{attribute 'linkalways'} 
{attribute 'no_explicit_call' := 'This FB is a CLASS and must be accessed using methods or properties'}
{attribute 'enable_dynamic_creation'}
FUNCTION_BLOCK _DWORD EXTENDS NumericDatatypeBase implements I_DWORD
VAR
	localData : DWORD;
	activeData : REFERENCE TO DWORD REF= localData;
END_VAR

PROPERTY PUBLIC Address : PVOID
GET
Address := ADR(activeData);
END_GET
END_PROPERTY

METHOD PUBLIC ClearReference
VAR_INPUT
END_VAR
activeData REF= localData;
END_METHOD

METHOD PUBLIC Clone : I_Datatype
VAR
    pClone : POINTER TO _DWORD;
END_VAR
pClone := __NEW(_DWORD(InitialValue := Value));
Clone := pClone^;
END_METHOD

METHOD FB_init : BOOL
VAR_INPUT
	bInitRetains : BOOL; // if TRUE, the retain variables are initialized (warm start / cold start)
	bInCopyCode : BOOL;  // if TRUE, the instance afterwards gets moved WORDo the copy code (online change)
	InitialValue : DWORD;
END_VAR
localData := InitialValue;
END_METHOD

PROPERTY PUBLIC IsEven : BOOL
GET
IsEven := (Value mod 2) = 0;
END_GET
END_PROPERTY

PROPERTY PUBLIC IsFloat : BOOL
GET
IsFloat := FALSE;
END_GET
END_PROPERTY

PROPERTY PUBLIC IsSigned : BOOL
GET
IsSigned := FALSE;
END_GET
END_PROPERTY

METHOD PUBLIC MakeReferenceTo
VAR_INPUT
	ReferenceTarget : REFERENCE TO DWORD;
END_VAR
activeData REF= ReferenceTarget;
END_METHOD

PROPERTY PUBLIC MaxValue : DWORD
GET
MaxValue := DatatypeLimits.DWORD_MAX_VALUE;
END_GET
END_PROPERTY

PROPERTY PUBLIC MinValue : DWORD
GET
MinValue := DatatypeLimits.DWORD_MIN_VALUE;
END_GET
END_PROPERTY

METHOD PROTECTED SerializeMaxValue
VAR_INPUT
	Serializer : I_Serializer;
END_VAR
Serializer.AddDword(MaxValue);
END_METHOD

METHOD PROTECTED SerializeMinValue
VAR_INPUT
	Serializer : I_Serializer;
END_VAR
Serializer.AddDword(MinValue);
END_METHOD

METHOD PUBLIC SerializeWith
VAR_INPUT
	Serializer : I_Serializer;
END_VAR
Serializer.AddDword(activeData);
END_METHOD

PROPERTY PUBLIC Size : UDINT
GET
Size := SIZEOF(activeData);
END_GET
END_PROPERTY

METHOD PUBLIC TryConvertTo : BOOL
VAR_INPUT
	Destination : ANY;
END_VAR
TryConvertTo := TryConvert_DWORD_To_Destination(activeData, Destination);
END_METHOD

METHOD PUBLIC TryConvertTo_ : BOOL
VAR_INPUT
	Destination : I_Datatype;
END_VAR
VAR
	resultofBitConversion : BOOL;
	destinationAs_BIT : I_BIT;
	destinationAs_BOOL : I_BOOL;
	destinationAs_BYTE : I_BYTE;
	destinationAs_DINT : I_DINT;
	destinationAs_DT : I_DT;
	destinationAs_DWORD : I_DWORD;
	destinationAs_INT : I_INT;
	destinationAs_LINT : I_LINT;
	destinationAs_LREAL : I_LREAL;
	destinationAs_LWORD : I_LWORD;
	destinationAs_REAL : I_REAL;
	destinationAs_SINT : I_SINT;
	destinationAs_STRING : I_STRING;
	destinationAs_TOD : I_TOD;
	destinationAs_UDINT : I_UDINT;
	destinationAs_UINT : I_UINT;
	destinationAs_ULINT : I_ULINT;
	destinationAs_USINT : I_USINT;
	destinationAs_WORD : I_WORD;
END_VAR
IF destination.TryResolveAs_BIT(destinationAs_BIT) AND_THEN TryConvert_DWORD_TO_BOOL(activeData, resultofBitConversion) THEN
	destinationAs_BIT.Value := resultOfBitConversion;
	TryConvertTo_ := TRUE;
	RETURN;
END_IF

IF destination.TryResolveAs_BOOL(destinationAs_BOOL) THEN
	TryConvertTo_ := TryConvert_DWORD_TO_BOOL(activeData, destinationAs_BOOL.Value);
	RETURN;
END_IF
		
IF destination.TryResolveAs_BYTE(destinationAs_BYTE) THEN
	TryConvertTo_ := TryConvert_DWORD_TO_BYTE(activeData, destinationAs_BYTE.Value);
	RETURN;
END_IF

IF destination.TryResolveAs_DINT(destinationAs_DINT) THEN
	TryConvertTo_ := TryConvert_DWORD_TO_DINT(activeData, destinationAs_DINT.Value);
	RETURN;
END_IF

IF destination.TryResolveAs_DT(destinationAs_DT) THEN
	TryConvertTo_ := TryConvert_DWORD_TO_DT(activeData, destinationAs_DT.Value);
	RETURN;
END_IF

IF destination.TryResolveAs_DWORD(destinationAs_DWORD) THEN
	TryConvertTo_ := TryConvert_DWORD_TO_DWORD(activeData, destinationAs_DWORD.Value);
	RETURN;
END_IF

IF destination.TryResolveAs_INT(destinationAs_INT) THEN
	TryConvertTo_ := TryConvert_DWORD_TO_INT(activeData, destinationAs_INT.Value);
	RETURN;
END_IF

IF destination.TryResolveAs_LINT(destinationAs_LINT) THEN
	TryConvertTo_ := TryConvert_DWORD_TO_LINT(activeData, destinationAs_LINT.Value);
	RETURN;
END_IF

IF destination.TryResolveAs_LREAL(destinationAs_LREAL) THEN
	TryConvertTo_ := TryConvert_DWORD_TO_LREAL(activeData, destinationAs_LREAL.Value);
	RETURN;
END_IF

IF destination.TryResolveAs_LWORD(destinationAs_LWORD) THEN
	TryConvertTo_ := TryConvert_DWORD_TO_LWORD(activeData, destinationAs_LWORD.Value);
	RETURN;
END_IF

IF destination.TryResolveAs_REAL(destinationAs_REAL) THEN
	TryConvertTo_ := TryConvert_DWORD_TO_REAL(activeData, destinationAs_REAL.Value);
	RETURN;
END_IF

IF destination.TryResolveAs_SINT(destinationAs_SINT) THEN
	TryConvertTo_ := TryConvert_DWORD_TO_SINT(activeData, destinationAs_SINT.Value);
	RETURN;
END_IF

IF destination.TryResolveAs_STRING(destinationAs_STRING) THEN
	TryConvertTo_ := TryConvert_DWORD_TO_STRING(activeData, destinationAs_STRING.Value);
	RETURN;
END_IF

IF destination.TryResolveAs_TOD(destinationAs_TOD) THEN
	TryConvertTo_ := TryConvert_DWORD_TO_TOD(activeData, destinationAs_TOD.Value);
	RETURN;
END_IF

IF destination.TryResolveAs_UDINT(destinationAs_UDINT) THEN
	TryConvertTo_ := TryConvert_DWORD_TO_UDINT(activeData, destinationAs_UDINT.Value);
	RETURN;
END_IF

IF destination.TryResolveAs_UINT(destinationAs_UINT) THEN
	TryConvertTo_ := TryConvert_DWORD_TO_UINT(activeData, destinationAs_UINT.Value);
	RETURN;
END_IF

IF destination.TryResolveAs_ULINT(destinationAs_ULINT) THEN
	TryConvertTo_ := TryConvert_DWORD_TO_ULINT(activeData, destinationAs_ULINT.Value);
	RETURN;
END_IF

IF destination.TryResolveAs_USINT(destinationAs_USINT) THEN
	TryConvertTo_ := TryConvert_DWORD_TO_USINT(activeData, destinationAs_USINT.Value);
	RETURN;
END_IF

IF destination.TryResolveAs_WORD(destinationAs_WORD) THEN
	TryConvertTo_ := TryConvert_DWORD_TO_WORD(activeData, destinationAs_WORD.Value);
	RETURN;
END_IF
END_METHOD

METHOD TryDeserializeFrom : BOOL
VAR_INPUT
	Deserializer : I_Deserializer;
	Feedback : I_DeserializerFeedback;
END_VAR
TryDeserializeFrom := Deserializer.TryGetDword(activeData, Feedback);
END_METHOD

METHOD TryMakeReferenceTo : BOOL
VAR_INPUT
	Target : I_Datatype;
END_VAR
VAR
	pTargetData : POINTER TO DWORD;
END_VAR
IF NOT IsEquivalentTo(Target) THEN
	RETURN;
END_IF

pTargetData := Target.Address;
activeData REF= pTargetData^;
TryMakeReferenceTo := TRUE;
END_METHOD

METHOD PUBLIC TryResolveAs_DWORD : BOOL
VAR_INPUT
	Destination : REFERENCE TO I_DWORD;
END_VAR
Destination := THIS^;
TryResolveAs_DWORD := TRUE;
END_METHOD

PROPERTY PUBLIC TypeName : T_MAXSTRING
GET
TypeName := 'DWORD';
END_GET
END_PROPERTY

PROPERTY PUBLIC Value : REFERENCE TO DWORD
GET
Value REF= activeData;
END_GET
END_PROPERTY

END_FUNCTION_BLOCK

(* stored: Version 1.1.0.1, ProductVersion 3.1.4024.15
   POU _DWORD: Id {0e1f4684-9ced-429c-808b-7eae4b4c544d}, SpecialFunc None
   Folder Constructor: Id {ed0f11a9-1e9f-4982-8f38-38243a563b64}
   Folder Protected: Id {81979a9d-08ab-4990-a6a1-6d8257d387e2}
   Property Address: Id {db5664d4-745e-4039-a24f-c4ccfecba779}
   Get Get: Id {e031636d-09ee-4c01-a84d-b6877667d967}
   Method ClearReference: Id {d4461140-18cc-4879-b0d4-8191674e6247}
   Method Clone: Id {94d3bddf-8fcb-4938-8fbd-23c2da87ed5a}
   Method FB_init: Id {12a44695-f484-4b13-adf1-9bfc8d3ddbe4}
   Property IsEven: Id {a9233086-77fa-0502-3db7-4b000f1aa9c4}
   Get Get: Id {42c8b3e7-f556-0983-013b-60f8adaee327}
   Property IsFloat: Id {ad06f207-ab0a-4f8c-a31f-a02263d34b51}
   Get Get: Id {203ea2a5-3922-43d2-862b-de05e5f89dd5}
   Property IsSigned: Id {513f9891-7111-4f35-92cb-cbc81f2c7472}
   Get Get: Id {8417e378-9fc5-4222-8e5d-eb450dda174b}
   Method MakeReferenceTo: Id {8fdcbcd4-27ca-44db-b8f8-fc8112ae5937}
   Property MaxValue: Id {034a1662-e6c7-4cbe-a2fc-aea858209350}
   Get Get: Id {81b19176-2120-431f-8056-dc7df3b20cc4}
   Property MinValue: Id {4ec11c32-e180-4d34-a9a0-1335281bd831}
   Get Get: Id {17477731-f195-44fc-b396-e42b5f51c8cc}
   Method SerializeMaxValue: Id {75a91e09-dc3c-4443-9fe4-2d3f65219af9}
   Method SerializeMinValue: Id {22897b76-1a27-4528-a271-d22b15e82d34}
   Method SerializeWith: Id {a9225849-74b7-48d0-a560-79fcd6fd118e}
   Property Size: Id {894da6f1-f132-4366-ac78-06d64875cba0}
   Get Get: Id {d861d9bb-218c-495e-99c8-0b207d9f8e67}
   Method TryConvertTo: Id {0bd32bb8-2a5f-04d7-38cb-a5770b81db39}
   Method TryConvertTo_: Id {e866a366-9f80-0d7b-2ed9-934ed139960c}
   Method TryDeserializeFrom: Id {83d5ad43-9e13-4e41-a478-5b9183f3167e}
   Method TryMakeReferenceTo: Id {4324d9f8-185a-44d1-9234-d6ed4995ead4}
   Method TryResolveAs_DWORD: Id {993b2d78-9268-06cf-1f4c-9a283c0b4ade}
   Property TypeName: Id {6f2720f4-af59-4d51-907f-292473cf57e7}
   Get Get: Id {7be10ba1-1f8b-4a60-8722-76feada590bc}
   Property Value: Id {fdccc3f4-cdf6-4251-a895-2c5af3829da4}
   Get Get: Id {393439f2-f918-4cc0-a08a-023c84afe948} *)
